PROGRAM HMI
VAR_INPUT
	BMS_Display				: BAT_NARADA;
	PCS_Display				: PCS_Sma;
	ESS_Display 			: ESS_Exd;
	
	PTR_Display				: PTR_Exd;
	INV_Display				: INV_Huawei;
	
END_VAR

// HPP
	HPP_HMI();
	
	BESS_HMI();
	
	SPP_HMI();

METHOD M_UserManagement : BOOL
VAR_INPUT
END_VAR
END_METHOD

END_PROGRAM

(* stored: Version 1.1.0.1, ProductVersion 3.1.4024.12
   POU HMI: Id {6d01684d-6c73-4991-ab6c-aac9e62c35d7}, SpecialFunc None
   Method M_UserManagement: Id {6cb76ec5-7d1f-45f7-b294-0686a4d23b9e} *)
